// TIA Portal V17 export
// export: Created 2022-07-20T07:02:30.2040415Z, ExportSetting WithDefaults, DisplayName Totally Integrated Automation Portal, DisplayVersion V17, DisplayName TIA Portal Openness, DisplayVersion V17, DisplayName TIA Portal Version Control Interface, DisplayVersion V17, DisplayName SINAMICS Startdrive Advanced, DisplayVersion V17, DisplayName SINAMICS Startdrive G130, G150, S120, S150, SINAMICS MV, S210, DisplayVersion V17, DisplayName SINAMICS Startdrive G110M, G120, G120C, G120D, G120P, G115D, DisplayVersion V17, DisplayName STEP 7 Professional, DisplayVersion V17, DisplayName STEP 7 Safety, DisplayVersion V17, DisplayName WinCC Advanced, DisplayVersion V17
FUNCTION_BLOCK "FB11000_SynchronousAxis"   // FB11000, LAD
TITLE = Manage positioning axis
{ S7_Optimized_Access := 'TRUE' }
VERSION : 0.1
// stored: AutoNumber false, IsIECCheckEnabled false, IsRetainMemResEnabled false, MemoryReserve 100, SetENOAutomatically false, UDAEnableTagReadback false
   VAR_INPUT
      Cam : DB_ANY;
   END_VAR
   VAR_IN_OUT
      Axis : TO_SynchronousAxis;   // Reference to axis to be controlled
      Master : TO_Axis;
      Interface : "stAxis";
   END_VAR
   VAR
      instLAxisCtrl_GetAxisStatusWord : "LAxisCtrl_GetAxisStatusWord";
      instLAxisCtrl_Axis { S7_SetPoint := 'True'} : "LAxisCtrl_SyncAxisCamming";
      instLAxisCtrl_AxisWarningWord { S7_SetPoint := 'True'} : "LAxisCtrl_GetAxisWarningWord";
      instLAxisCtrl_AxisErrorWord { S7_SetPoint := 'True'} : "LAxisCtrl_GetAxisErrorWord";
   END_VAR
   VAR_TEMP   // added for the SCL form of the ladder/FBD networks
      _w1 : Bool;
   END_VAR
BEGIN

REGION Network 1 (SCL): Comments
   //==========================================================================================
   // SIEMENS SAS      RC-FR DI FA APC
   //------------------------------------------------------------------------------------------
   // Restrictions:    TIA V16 and more
   // Requirements:    S7-1500T + LAxisCtrl library
   // Functionality:   This function block offers basic functionalities for TO SynchronousAxis
   //                  Based on LCtrlAxis_PosAxis with additionnal functionality
   //------------------------------------------------------------------------------------------
   // Change log table:
   // Version      Date        Expert in charge    Changes applied
   // 01.00.01     09.06.2020  RTO                 First released version
   //==========================================================================================
END_REGION

REGION Network 2: Manage axis functions
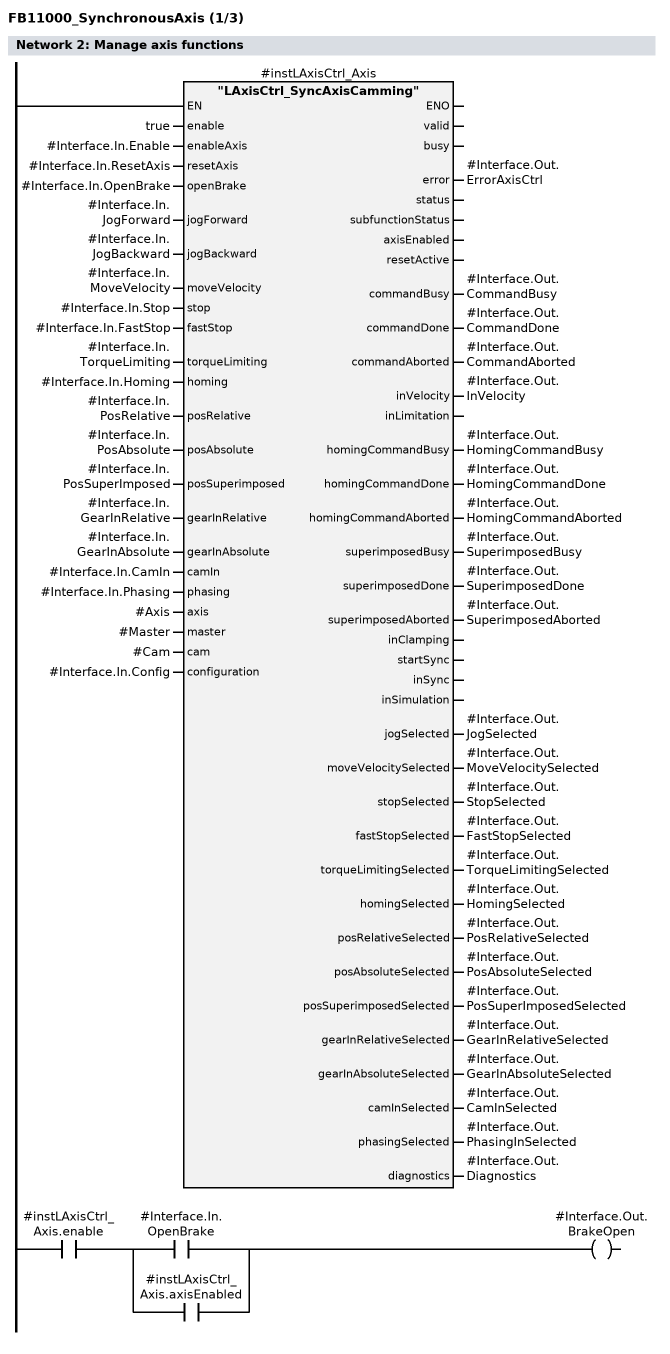
   RUNG wire#powerrail
      #instLAxisCtrl_Axis(enable := true, enableAxis := #Interface.In.Enable, resetAxis := #Interface.In.ResetAxis, openBrake := #Interface.In.OpenBrake, jogForward := #Interface.In.JogForward, jogBackward := #Interface.In.JogBackward, moveVelocity := #Interface.In.MoveVelocity, stop := #Interface.In.Stop, fastStop := #Interface.In.FastStop, torqueLimiting := #Interface.In.TorqueLimiting, homing := #Interface.In.Homing, posRelative := #Interface.In.PosRelative, posAbsolute := #Interface.In.PosAbsolute, posSuperimposed := #Interface.In.PosSuperImposed, gearInRelative := #Interface.In.GearInRelative, gearInAbsolute := #Interface.In.GearInAbsolute, camIn := #Interface.In.CamIn, phasing := #Interface.In.Phasing, axis := #Axis, master := #Master, cam := #Cam, configuration := #Interface.In.Config, valid =>, busy =>, error => #Interface.Out.ErrorAxisCtrl, status =>, subfunctionStatus =>, axisEnabled =>, resetActive =>, commandBusy => #Interface.Out.CommandBusy, commandDone => #Interface.Out.CommandDone, commandAborted => #Interface.Out.CommandAborted, inVelocity => #Interface.Out.InVelocity, inLimitation =>, homingCommandBusy => #Interface.Out.HomingCommandBusy, homingCommandDone => #Interface.Out.HomingCommandDone, homingCommandAborted => #Interface.Out.HomingCommandAborted, superimposedBusy => #Interface.Out.SuperimposedBusy, superimposedDone => #Interface.Out.SuperimposedDone, superimposedAborted => #Interface.Out.SuperimposedAborted, inClamping =>, startSync =>, inSync =>, inSimulation =>, jogSelected => #Interface.Out.JogSelected, moveVelocitySelected => #Interface.Out.MoveVelocitySelected, stopSelected => #Interface.Out.StopSelected, fastStopSelected => #Interface.Out.FastStopSelected, torqueLimitingSelected => #Interface.Out.TorqueLimitingSelected, homingSelected => #Interface.Out.HomingSelected, posRelativeSelected => #Interface.Out.PosRelativeSelected, posAbsoluteSelected => #Interface.Out.PosAbsoluteSelected, posSuperimposedSelected => #Interface.Out.PosSuperImposedSelected, gearInRelativeSelected => #Interface.Out.GearInRelativeSelected, gearInAbsoluteSelected => #Interface.Out.GearInAbsoluteSelected, camInSelected => #Interface.Out.CamInSelected, phasingSelected => #Interface.Out.PhasingInSelected, diagnostics => #Interface.Out.Diagnostics)
   END_RUNG
   RUNG wire#powerrail
      Contact( #instLAxisCtrl_Axis.enable )
      wire#w1
      Contact( #Interface.In.OpenBrake )
      wire#w2
      Coil( #Interface.Out.BrakeOpen )
   END_RUNG
   RUNG wire#w1
      Contact( #instLAxisCtrl_Axis.axisEnabled )
   END_RUNG wire#w2
   // the same network as SCL:
   #instLAxisCtrl_Axis(enable := true,   // "LAxisCtrl_SyncAxisCamming"
                       enableAxis := #Interface.In.Enable,
                       resetAxis := #Interface.In.ResetAxis,
                       openBrake := #Interface.In.OpenBrake,
                       jogForward := #Interface.In.JogForward,
                       jogBackward := #Interface.In.JogBackward,
                       moveVelocity := #Interface.In.MoveVelocity,
                       stop := #Interface.In.Stop,
                       fastStop := #Interface.In.FastStop,
                       torqueLimiting := #Interface.In.TorqueLimiting,
                       homing := #Interface.In.Homing,
                       posRelative := #Interface.In.PosRelative,
                       posAbsolute := #Interface.In.PosAbsolute,
                       posSuperimposed := #Interface.In.PosSuperImposed,
                       gearInRelative := #Interface.In.GearInRelative,
                       gearInAbsolute := #Interface.In.GearInAbsolute,
                       camIn := #Interface.In.CamIn,
                       phasing := #Interface.In.Phasing,
                       axis := #Axis,
                       master := #Master,
                       cam := #Cam,
                       configuration := #Interface.In.Config,
                       error => #Interface.Out.ErrorAxisCtrl,
                       commandBusy => #Interface.Out.CommandBusy,
                       commandDone => #Interface.Out.CommandDone,
                       commandAborted => #Interface.Out.CommandAborted,
                       inVelocity => #Interface.Out.InVelocity,
                       homingCommandBusy => #Interface.Out.HomingCommandBusy,
                       homingCommandDone => #Interface.Out.HomingCommandDone,
                       homingCommandAborted => #Interface.Out.HomingCommandAborted,
                       superimposedBusy => #Interface.Out.SuperimposedBusy,
                       superimposedDone => #Interface.Out.SuperimposedDone,
                       superimposedAborted => #Interface.Out.SuperimposedAborted,
                       jogSelected => #Interface.Out.JogSelected,
                       moveVelocitySelected => #Interface.Out.MoveVelocitySelected,
                       stopSelected => #Interface.Out.StopSelected,
                       fastStopSelected => #Interface.Out.FastStopSelected,
                       torqueLimitingSelected => #Interface.Out.TorqueLimitingSelected,
                       homingSelected => #Interface.Out.HomingSelected,
                       posRelativeSelected => #Interface.Out.PosRelativeSelected,
                       posAbsoluteSelected => #Interface.Out.PosAbsoluteSelected,
                       posSuperimposedSelected => #Interface.Out.PosSuperImposedSelected,
                       gearInRelativeSelected => #Interface.Out.GearInRelativeSelected,
                       gearInAbsoluteSelected => #Interface.Out.GearInAbsoluteSelected,
                       camInSelected => #Interface.Out.CamInSelected,
                       phasingSelected => #Interface.Out.PhasingInSelected,
                       diagnostics => #Interface.Out.Diagnostics);
   #Interface.Out.BrakeOpen := #instLAxisCtrl_Axis.enable AND (#Interface.In.OpenBrake OR #instLAxisCtrl_Axis.axisEnabled);
END_REGION

REGION Network 3: Get axis status word
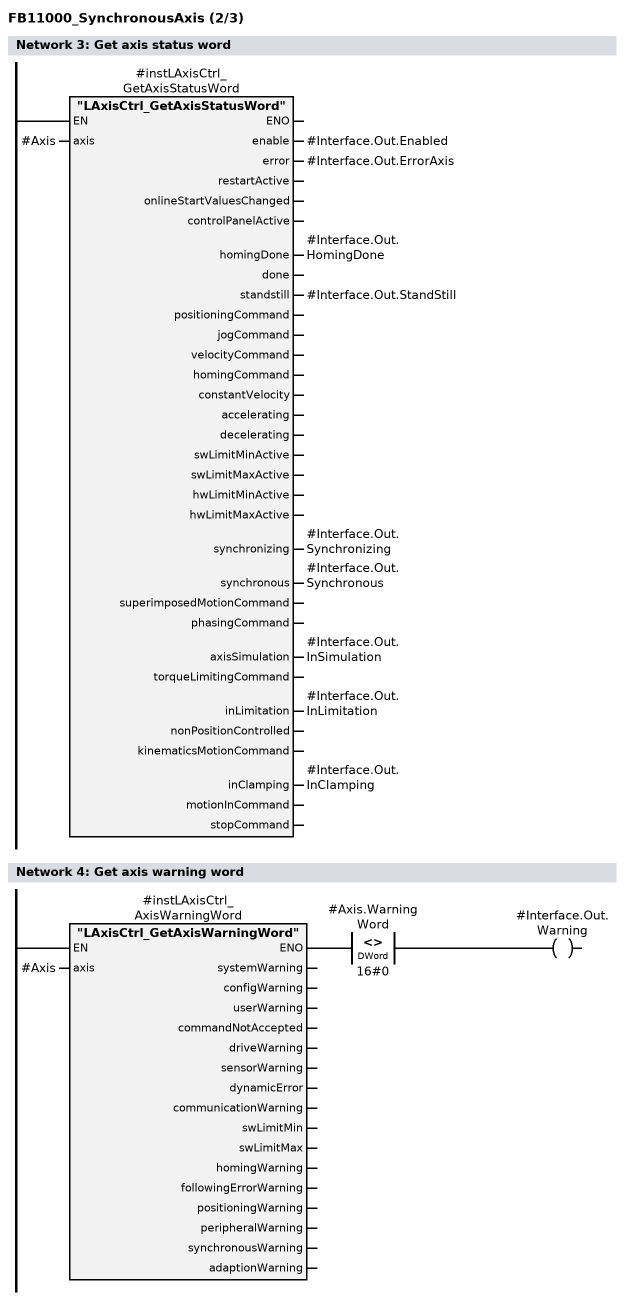
   RUNG wire#powerrail
      #instLAxisCtrl_GetAxisStatusWord(axis := #Axis, enable => #Interface.Out.Enabled, error => #Interface.Out.ErrorAxis, restartActive =>, onlineStartValuesChanged =>, controlPanelActive =>, homingDone => #Interface.Out.HomingDone, done =>, standstill => #Interface.Out.StandStill, positioningCommand =>, jogCommand =>, velocityCommand =>, homingCommand =>, constantVelocity =>, accelerating =>, decelerating =>, swLimitMinActive =>, swLimitMaxActive =>, hwLimitMinActive =>, hwLimitMaxActive =>, synchronizing => #Interface.Out.Synchronizing, synchronous => #Interface.Out.Synchronous, superimposedMotionCommand =>, phasingCommand =>, axisSimulation => #Interface.Out.InSimulation, torqueLimitingCommand =>, inLimitation => #Interface.Out.InLimitation, nonPositionControlled =>, kinematicsMotionCommand =>, inClamping => #Interface.Out.InClamping, motionInCommand =>, stopCommand =>)
   END_RUNG
   // the same network as SCL:
   #instLAxisCtrl_GetAxisStatusWord(axis := #Axis,   // "LAxisCtrl_GetAxisStatusWord"
                           enable => #Interface.Out.Enabled,
                           error => #Interface.Out.ErrorAxis,
                           homingDone => #Interface.Out.HomingDone,
                           standstill => #Interface.Out.StandStill,
                           synchronizing => #Interface.Out.Synchronizing,
                           synchronous => #Interface.Out.Synchronous,
                           axisSimulation => #Interface.Out.InSimulation,
                           inLimitation => #Interface.Out.InLimitation,
                           inClamping => #Interface.Out.InClamping);
END_REGION

REGION Network 4: Get axis warning word
   RUNG wire#powerrail
      #instLAxisCtrl_AxisWarningWord(axis := #Axis, systemWarning =>, configWarning =>, userWarning =>, commandNotAccepted =>, driveWarning =>, sensorWarning =>, dynamicError =>, communicationWarning =>, swLimitMin =>, swLimitMax =>, homingWarning =>, followingErrorWarning =>, positioningWarning =>, peripheralWarning =>, synchronousWarning =>, adaptionWarning =>)
      { S7_Templates := "SrcType := DWord" } NE_Contact(in1 := #Axis.WarningWord, in2 := 16#0)
      Coil( #Interface.Out.Warning )
   END_RUNG
   // the same network as SCL:
   #instLAxisCtrl_AxisWarningWord(axis := #Axis, ENO => #_w1);   // "LAxisCtrl_GetAxisWarningWord"
   #Interface.Out.Warning := #_w1 AND (#Axis.WarningWord <> 16#0);
END_REGION

REGION Network 5: Get axis error word
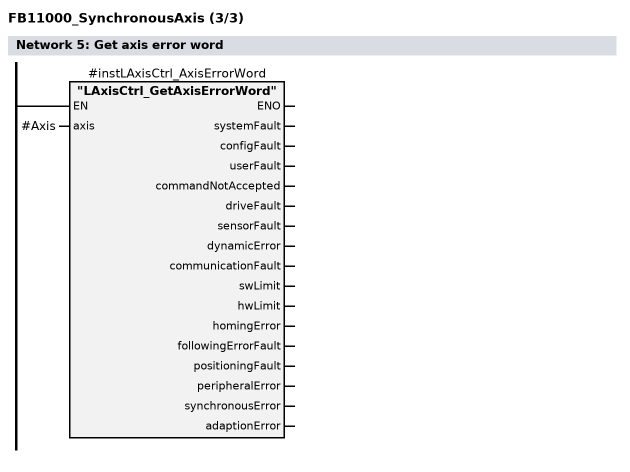
   RUNG wire#powerrail
      #instLAxisCtrl_AxisErrorWord(axis := #Axis, systemFault =>, configFault =>, userFault =>, commandNotAccepted =>, driveFault =>, sensorFault =>, dynamicError =>, communicationFault =>, swLimit =>, hwLimit =>, homingError =>, followingErrorFault =>, positioningFault =>, peripheralError =>, synchronousError =>, adaptionError =>)
   END_RUNG
   // the same network as SCL:
   #instLAxisCtrl_AxisErrorWord(axis := #Axis);   // "LAxisCtrl_GetAxisErrorWord"
END_REGION

REGION Network 6 (SCL): Get actual values of axis
   #Interface.Out.ActualPosition := #Axis.ActualPosition;
   #Interface.Out.ActualVelocity := #Axis.ActualVelocity;
   #Interface.Out.ActualAcceleration := #Axis.ActualAcceleration;

   #Interface.Out.ActualFollowingError := #Axis.StatusPositioning.FollowingError;
   #Interface.Out.ActualTorque := #Axis.StatusTorqueData.ActualTorque;
END_REGION
END_FUNCTION_BLOCK
